(* PLC project Unnamed, Unknown Unnamed 1 *)
(* stored: creationDateTime 2023-05-01T23:10:03, modificationDateTime 2023-05-08T22:46:58 *)

PROGRAM program0
  VAR
    EmStop AT %IX0.1 : BOOL;
    E1 AT %IX0.2 : BOOL;
    E2 AT %IX0.3 : BOOL;
    P1 AT %QX0.0 : BOOL;
    P2 AT %QX0.1 : BOOL;
  END_VAR

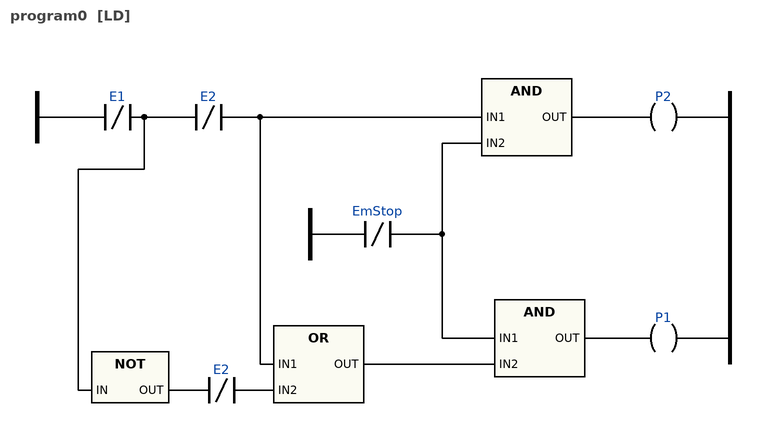
(* LD diagram, written out as Structured Text *)
P2 := NOT E1 AND NOT E2 AND NOT EmStop;
P1 := NOT EmStop AND (NOT E1 AND NOT E2 OR NOT (NOT E1) AND NOT E2);
END_PROGRAM

CONFIGURATION Config0
  RESOURCE Res0 ON PLC
    TASK task0(INTERVAL := T#20ms, PRIORITY := 0);
    PROGRAM instance0 WITH task0 : program0;
  END_RESOURCE
END_CONFIGURATION
